FUNCTION_BLOCK joystick
VAR_INPUT
END_VAR
VAR_OUTPUT
END_VAR
VAR
END_VAR

END_FUNCTION_BLOCK

(* stored: Version 1.1.0.1, ProductVersion 3.1.4024.12
   POU joystick: Id {a5b1796a-d5de-409f-b15d-f3c0b8424381}, SpecialFunc None *)
